KUKA KRL program: exC126.src, exC126.dat

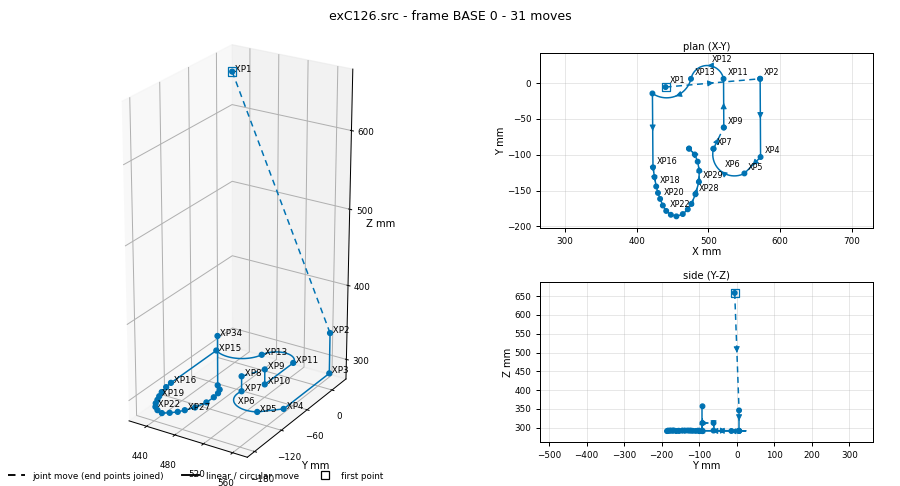
[picture p0: tool path of exC126.src in frame BASE 0, 31 of 33 moves have a stored position in this frame; points joined in program order, loops and branches not executed]
--- exC126.src ---
&ACCESS RVP
&REL 41
&PARAM EDITMASK = *
&PARAM TEMPLATE = C:\KRC\Roboter\Template\vorgabe
&PARAM DISKPATH = KRC:\R1\Program\126PARCIAL
DEF exC126( )
;FOLD INI;%{PE}
  ;FOLD BASISTECH INI
    GLOBAL INTERRUPT DECL 3 WHEN $STOPMESS==TRUE DO IR_STOPM ( )
    INTERRUPT ON 3
    BAS (#INITMOV,0 )
  ;ENDFOLD (BASISTECH INI)
  ;FOLD USER INI
    ;Make your modifications here

  ;ENDFOLD (USER INI)
;ENDFOLD (INI)

;FOLD SPTP HOME Vel=100 % DEFAULT ;%{PE}
;FOLD Parameters ;%{h}
;Params IlfProvider=kukaroboter.basistech.inlineforms.movement.spline; Kuka.IsGlobalPoint=False; Kuka.PointName=HOME; Kuka.BlendingEnabled=False; Kuka.MoveDataPtpName=DEFAULT; Kuka.VelocityPtp=100; Kuka.VelocityFieldEnabled=True; Kuka.CurrentCDSetIndex=0; Kuka.MovementParameterFieldEnabled=True; IlfCommand=SPTP
;ENDFOLD
SPTP XHOME WITH $VEL_AXIS[1] = SVEL_JOINT(100.0), $TOOL = STOOL2(FHOME), $BASE = SBASE(FHOME.BASE_NO), $IPO_MODE = SIPO_MODE(FHOME.IPO_FRAME), $LOAD = SLOAD(FHOME.TOOL_NO), $ACC_AXIS[1] = SACC_JOINT(PDEFAULT), $APO = SAPO_PTP(PDEFAULT), $GEAR_JERK[1] = SGEAR_JERK(PDEFAULT), $COLLMON_TOL_PRO[1] = USE_CM_PRO_VALUES(0)
;ENDFOLD

;FOLD SPTP P1 Vel=100 % PDAT1 Tool[1]:SMC Base[0] ;%{PE}
;FOLD Parameters ;%{h}
;Params IlfProvider=kukaroboter.basistech.inlineforms.movement.spline; Kuka.IsGlobalPoint=False; Kuka.PointName=P1; Kuka.BlendingEnabled=False; Kuka.MoveDataPtpName=PDAT1; Kuka.VelocityPtp=100; Kuka.VelocityFieldEnabled=True; Kuka.ColDetectFieldEnabled=True; Kuka.CurrentCDSetIndex=0; Kuka.MovementParameterFieldEnabled=True; IlfCommand=SPTP
;ENDFOLD
SPTP XP1 WITH $VEL_AXIS[1] = SVEL_JOINT(100.0), $TOOL = STOOL2(FP1), $BASE = SBASE(FP1.BASE_NO), $IPO_MODE = SIPO_MODE(FP1.IPO_FRAME), $LOAD = SLOAD(FP1.TOOL_NO), $ACC_AXIS[1] = SACC_JOINT(PPDAT1), $APO = SAPO_PTP(PPDAT1), $GEAR_JERK[1] = SGEAR_JERK(PPDAT1), $COLLMON_TOL_PRO[1] = USE_CM_PRO_VALUES(0)
;ENDFOLD
;FOLD SPTP P2 Vel=100 % PDAT2 Tool[1]:SMC Base[0] ;%{PE}
;FOLD Parameters ;%{h}
;Params IlfProvider=kukaroboter.basistech.inlineforms.movement.spline; Kuka.IsGlobalPoint=False; Kuka.PointName=P2; Kuka.BlendingEnabled=False; Kuka.MoveDataPtpName=PDAT2; Kuka.VelocityPtp=100; Kuka.VelocityFieldEnabled=True; Kuka.ColDetectFieldEnabled=True; Kuka.CurrentCDSetIndex=0; Kuka.MovementParameterFieldEnabled=True; IlfCommand=SPTP
;ENDFOLD
SPTP XP2 WITH $VEL_AXIS[1] = SVEL_JOINT(100.0), $TOOL = STOOL2(FP2), $BASE = SBASE(FP2.BASE_NO), $IPO_MODE = SIPO_MODE(FP2.IPO_FRAME), $LOAD = SLOAD(FP2.TOOL_NO), $ACC_AXIS[1] = SACC_JOINT(PPDAT2), $APO = SAPO_PTP(PPDAT2), $GEAR_JERK[1] = SGEAR_JERK(PPDAT2), $COLLMON_TOL_PRO[1] = USE_CM_PRO_VALUES(0)
;ENDFOLD
;FOLD SLIN P3 Vel=2 m/s CPDAT1 Tool[1]:SMC Base[0] ;%{PE}
;FOLD Parameters ;%{h}
;Params IlfProvider=kukaroboter.basistech.inlineforms.movement.spline; Kuka.IsGlobalPoint=False; Kuka.PointName=P3; Kuka.BlendingEnabled=False; Kuka.MoveDataName=CPDAT1; Kuka.VelocityPath=2; Kuka.VelocityFieldEnabled=True; Kuka.ColDetectFieldEnabled=True; Kuka.CurrentCDSetIndex=0; Kuka.MovementParameterFieldEnabled=True; IlfCommand=SLIN
;ENDFOLD
SLIN XP3 WITH $VEL = SVEL_CP(2.0, , LCPDAT1), $TOOL = STOOL2(FP3), $BASE = SBASE(FP3.BASE_NO), $IPO_MODE = SIPO_MODE(FP3.IPO_FRAME), $LOAD = SLOAD(FP3.TOOL_NO), $ACC = SACC_CP(LCPDAT1), $ORI_TYPE = SORI_TYP(LCPDAT1), $APO = SAPO(LCPDAT1), $JERK = SJERK(LCPDAT1), $COLLMON_TOL_PRO[1] = USE_CM_PRO_VALUES(0)
;ENDFOLD
;FOLD SLIN P4 Vel=2 m/s CPDAT2 Tool[1]:SMC Base[0] ;%{PE}
;FOLD Parameters ;%{h}
;Params IlfProvider=kukaroboter.basistech.inlineforms.movement.spline; Kuka.IsGlobalPoint=False; Kuka.PointName=P4; Kuka.BlendingEnabled=False; Kuka.MoveDataName=CPDAT2; Kuka.VelocityPath=2; Kuka.VelocityFieldEnabled=True; Kuka.ColDetectFieldEnabled=True; Kuka.CurrentCDSetIndex=0; Kuka.MovementParameterFieldEnabled=True; IlfCommand=SLIN
;ENDFOLD
SLIN XP4 WITH $VEL = SVEL_CP(2.0, , LCPDAT2), $TOOL = STOOL2(FP4), $BASE = SBASE(FP4.BASE_NO), $IPO_MODE = SIPO_MODE(FP4.IPO_FRAME), $LOAD = SLOAD(FP4.TOOL_NO), $ACC = SACC_CP(LCPDAT2), $ORI_TYPE = SORI_TYP(LCPDAT2), $APO = SAPO(LCPDAT2), $JERK = SJERK(LCPDAT2), $COLLMON_TOL_PRO[1] = USE_CM_PRO_VALUES(0)
;ENDFOLD
;FOLD SLIN P5 Vel=2 m/s CPDAT3 Tool[1]:SMC Base[0] ;%{PE}
;FOLD Parameters ;%{h}
;Params IlfProvider=kukaroboter.basistech.inlineforms.movement.spline; Kuka.IsGlobalPoint=False; Kuka.PointName=P5; Kuka.BlendingEnabled=False; Kuka.MoveDataName=CPDAT3; Kuka.VelocityPath=2; Kuka.VelocityFieldEnabled=True; Kuka.ColDetectFieldEnabled=True; Kuka.CurrentCDSetIndex=0; Kuka.MovementParameterFieldEnabled=True; IlfCommand=SLIN
;ENDFOLD
SLIN XP5 WITH $VEL = SVEL_CP(2.0, , LCPDAT3), $TOOL = STOOL2(FP5), $BASE = SBASE(FP5.BASE_NO), $IPO_MODE = SIPO_MODE(FP5.IPO_FRAME), $LOAD = SLOAD(FP5.TOOL_NO), $ACC = SACC_CP(LCPDAT3), $ORI_TYPE = SORI_TYP(LCPDAT3), $APO = SAPO(LCPDAT3), $JERK = SJERK(LCPDAT3), $COLLMON_TOL_PRO[1] = USE_CM_PRO_VALUES(0)
;ENDFOLD
;FOLD SCIRC P6 P7 Vel=2 m/s CPDAT4 Tool[1]:SMC Base[0] ;%{PE}
;FOLD Parameters ;%{h}
;Params IlfProvider=kukaroboter.basistech.inlineforms.movement.spline; Kuka.IsGlobalPoint=False; Kuka.PointName=P7; Kuka.HelpPointName=P6; Kuka.BlendingEnabled=False; Kuka.MoveDataName=CPDAT4; Kuka.VelocityPath=2; Kuka.VelocityFieldEnabled=True; Kuka.ColDetectFieldEnabled=True; Kuka.CurrentCDSetIndex=0; Kuka.MovementParameterFieldEnabled=True; IlfCommand=SCIRC
;ENDFOLD
SCIRC XP6, XP7 WITH $VEL = SVEL_CP(2.0, , LCPDAT4), $TOOL = STOOL2(FP7), $BASE = SBASE(FP7.BASE_NO), $IPO_MODE = SIPO_MODE(FP7.IPO_FRAME), $LOAD = SLOAD(FP7.TOOL_NO), $ACC = SACC_CP(LCPDAT4), $ORI_TYPE = SORI_TYP(LCPDAT4), $CIRC_TYPE = SCIRC_TYP(LCPDAT4), $APO = SAPO(LCPDAT4), $CIRC_MODE = SCIRC_M(LCPDAT4), $JERK = SJERK(LCPDAT4), $COLLMON_TOL_PRO[1] = USE_CM_PRO_VALUES(0)
;ENDFOLD
;FOLD SLIN P8 Vel=2 m/s CPDAT5 Tool[1]:SMC Base[0] ;%{PE}
;FOLD Parameters ;%{h}
;Params IlfProvider=kukaroboter.basistech.inlineforms.movement.spline; Kuka.IsGlobalPoint=False; Kuka.PointName=P8; Kuka.BlendingEnabled=False; Kuka.MoveDataName=CPDAT5; Kuka.VelocityPath=2; Kuka.VelocityFieldEnabled=True; Kuka.ColDetectFieldEnabled=True; Kuka.CurrentCDSetIndex=0; Kuka.MovementParameterFieldEnabled=True; IlfCommand=SLIN
;ENDFOLD
SLIN XP8 WITH $VEL = SVEL_CP(2.0, , LCPDAT5), $TOOL = STOOL2(FP8), $BASE = SBASE(FP8.BASE_NO), $IPO_MODE = SIPO_MODE(FP8.IPO_FRAME), $LOAD = SLOAD(FP8.TOOL_NO), $ACC = SACC_CP(LCPDAT5), $ORI_TYPE = SORI_TYP(LCPDAT5), $APO = SAPO(LCPDAT5), $JERK = SJERK(LCPDAT5), $COLLMON_TOL_PRO[1] = USE_CM_PRO_VALUES(0)
;ENDFOLD
;FOLD SPTP P9 Vel=100 % PDAT3 Tool[1]:SMC Base[0] ;%{PE}
;FOLD Parameters ;%{h}
;Params IlfProvider=kukaroboter.basistech.inlineforms.movement.spline; Kuka.IsGlobalPoint=False; Kuka.PointName=P9; Kuka.BlendingEnabled=False; Kuka.MoveDataPtpName=PDAT3; Kuka.VelocityPtp=100; Kuka.VelocityFieldEnabled=True; Kuka.ColDetectFieldEnabled=True; Kuka.CurrentCDSetIndex=0; Kuka.MovementParameterFieldEnabled=True; IlfCommand=SPTP
;ENDFOLD
SPTP XP9 WITH $VEL_AXIS[1] = SVEL_JOINT(100.0), $TOOL = STOOL2(FP9), $BASE = SBASE(FP9.BASE_NO), $IPO_MODE = SIPO_MODE(FP9.IPO_FRAME), $LOAD = SLOAD(FP9.TOOL_NO), $ACC_AXIS[1] = SACC_JOINT(PPDAT3), $APO = SAPO_PTP(PPDAT3), $GEAR_JERK[1] = SGEAR_JERK(PPDAT3), $COLLMON_TOL_PRO[1] = USE_CM_PRO_VALUES(0)
;ENDFOLD
;FOLD SLIN P10 Vel=2 m/s CPDAT6 Tool[1]:SMC Base[0] ;%{PE}
;FOLD Parameters ;%{h}
;Params IlfProvider=kukaroboter.basistech.inlineforms.movement.spline; Kuka.IsGlobalPoint=False; Kuka.PointName=P10; Kuka.BlendingEnabled=False; Kuka.MoveDataName=CPDAT6; Kuka.VelocityPath=2; Kuka.VelocityFieldEnabled=True; Kuka.ColDetectFieldEnabled=True; Kuka.CurrentCDSetIndex=0; Kuka.MovementParameterFieldEnabled=True; IlfCommand=SLIN
;ENDFOLD
SLIN XP10 WITH $VEL = SVEL_CP(2.0, , LCPDAT6), $TOOL = STOOL2(FP10), $BASE = SBASE(FP10.BASE_NO), $IPO_MODE = SIPO_MODE(FP10.IPO_FRAME), $LOAD = SLOAD(FP10.TOOL_NO), $ACC = SACC_CP(LCPDAT6), $ORI_TYPE = SORI_TYP(LCPDAT6), $APO = SAPO(LCPDAT6), $JERK = SJERK(LCPDAT6), $COLLMON_TOL_PRO[1] = USE_CM_PRO_VALUES(0)
;ENDFOLD
;FOLD SLIN P11 Vel=2 m/s CPDAT7 Tool[1]:SMC Base[0] ;%{PE}
;FOLD Parameters ;%{h}
;Params IlfProvider=kukaroboter.basistech.inlineforms.movement.spline; Kuka.IsGlobalPoint=False; Kuka.PointName=P11; Kuka.BlendingEnabled=False; Kuka.MoveDataName=CPDAT7; Kuka.VelocityPath=2; Kuka.VelocityFieldEnabled=True; Kuka.ColDetectFieldEnabled=True; Kuka.CurrentCDSetIndex=0; Kuka.MovementParameterFieldEnabled=True; IlfCommand=SLIN
;ENDFOLD
SLIN XP11 WITH $VEL = SVEL_CP(2.0, , LCPDAT7), $TOOL = STOOL2(FP11), $BASE = SBASE(FP11.BASE_NO), $IPO_MODE = SIPO_MODE(FP11.IPO_FRAME), $LOAD = SLOAD(FP11.TOOL_NO), $ACC = SACC_CP(LCPDAT7), $ORI_TYPE = SORI_TYP(LCPDAT7), $APO = SAPO(LCPDAT7), $JERK = SJERK(LCPDAT7), $COLLMON_TOL_PRO[1] = USE_CM_PRO_VALUES(0)
;ENDFOLD
;FOLD SCIRC P12 P13 Vel=2 m/s CPDAT8 Tool[1]:SMC Base[0] ;%{PE}
;FOLD Parameters ;%{h}
;Params IlfProvider=kukaroboter.basistech.inlineforms.movement.spline; Kuka.IsGlobalPoint=False; Kuka.PointName=P13; Kuka.HelpPointName=P12; Kuka.BlendingEnabled=False; Kuka.MoveDataName=CPDAT8; Kuka.VelocityPath=2; Kuka.VelocityFieldEnabled=True; Kuka.ColDetectFieldEnabled=True; Kuka.CurrentCDSetIndex=0; Kuka.MovementParameterFieldEnabled=True; IlfCommand=SCIRC
;ENDFOLD
SCIRC XP12, XP13 WITH $VEL = SVEL_CP(2.0, , LCPDAT8), $TOOL = STOOL2(FP13), $BASE = SBASE(FP13.BASE_NO), $IPO_MODE = SIPO_MODE(FP13.IPO_FRAME), $LOAD = SLOAD(FP13.TOOL_NO), $ACC = SACC_CP(LCPDAT8), $ORI_TYPE = SORI_TYP(LCPDAT8), $CIRC_TYPE = SCIRC_TYP(LCPDAT8), $APO = SAPO(LCPDAT8), $CIRC_MODE = SCIRC_M(LCPDAT8), $JERK = SJERK(LCPDAT8), $COLLMON_TOL_PRO[1] = USE_CM_PRO_VALUES(0)
;ENDFOLD
;FOLD SCIRC P14 P15 Vel=2 m/s CPDAT9 Tool[1]:SMC Base[0] ;%{PE}
;FOLD Parameters ;%{h}
;Params IlfProvider=kukaroboter.basistech.inlineforms.movement.spline; Kuka.IsGlobalPoint=False; Kuka.PointName=P15; Kuka.HelpPointName=P14; Kuka.BlendingEnabled=False; Kuka.MoveDataName=CPDAT9; Kuka.VelocityPath=2; Kuka.VelocityFieldEnabled=True; Kuka.ColDetectFieldEnabled=True; Kuka.CurrentCDSetIndex=0; Kuka.MovementParameterFieldEnabled=True; IlfCommand=SCIRC
;ENDFOLD
SCIRC XP14, XP15 WITH $VEL = SVEL_CP(2.0, , LCPDAT9), $TOOL = STOOL2(FP15), $BASE = SBASE(FP15.BASE_NO), $IPO_MODE = SIPO_MODE(FP15.IPO_FRAME), $LOAD = SLOAD(FP15.TOOL_NO), $ACC = SACC_CP(LCPDAT9), $ORI_TYPE = SORI_TYP(LCPDAT9), $CIRC_TYPE = SCIRC_TYP(LCPDAT9), $APO = SAPO(LCPDAT9), $CIRC_MODE = SCIRC_M(LCPDAT9), $JERK = SJERK(LCPDAT9), $COLLMON_TOL_PRO[1] = USE_CM_PRO_VALUES(0)
;ENDFOLD
;FOLD SLIN P16 Vel=2 m/s CPDAT10 Tool[1]:SMC Base[0] ;%{PE}
;FOLD Parameters ;%{h}
;Params IlfProvider=kukaroboter.basistech.inlineforms.movement.spline; Kuka.IsGlobalPoint=False; Kuka.PointName=P16; Kuka.BlendingEnabled=False; Kuka.MoveDataName=CPDAT10; Kuka.VelocityPath=2; Kuka.VelocityFieldEnabled=True; Kuka.ColDetectFieldEnabled=True; Kuka.CurrentCDSetIndex=0; Kuka.MovementParameterFieldEnabled=True; IlfCommand=SLIN
;ENDFOLD
SLIN XP16 WITH $VEL = SVEL_CP(2.0, , LCPDAT10), $TOOL = STOOL2(FP16), $BASE = SBASE(FP16.BASE_NO), $IPO_MODE = SIPO_MODE(FP16.IPO_FRAME), $LOAD = SLOAD(FP16.TOOL_NO), $ACC = SACC_CP(LCPDAT10), $ORI_TYPE = SORI_TYP(LCPDAT10), $APO = SAPO(LCPDAT10), $JERK = SJERK(LCPDAT10), $COLLMON_TOL_PRO[1] = USE_CM_PRO_VALUES(0)
;ENDFOLD
;FOLD SPLINE S1 Vel=2 m/s CPDAT11 Tool[1]:SMC Base[0] ;%{P} %CSPL_PARENT
;FOLD ;%{H}
;FOLD Parameters ;%{h}
;Params IlfProvider=kukaroboter.basistech.inlineforms.movement.splblock; Kuka.IsGlobalPoint=False; Kuka.SplineBlockPointName=S1; Kuka.BlendingEnabled=False; Kuka.MoveDataName=CPDAT11; Kuka.VelocityPath=2; Kuka.CurrentCDSetIndex=0; Kuka.MovementParameterFieldEnabled=True
;ENDFOLD
SPLINE WITH $VEL = SVEL_CP(2.0, , LCPDAT11), $TOOL = STOOL2(FS1), $BASE = SBASE(FS1.BASE_NO), $IPO_MODE = SIPO_MODE(FS1.IPO_FRAME), $LOAD = SLOAD(FS1.TOOL_NO), $ACC = SACC_CP(LCPDAT11), $APO = SAPO(LCPDAT11), $ORI_TYPE = SORI_TYP(LCPDAT11), $CIRC_TYPE = SCIRC_TYP(LCPDAT11), $JERK = SJERK(LCPDAT11), $COLLMON_TOL_PRO[1] = USE_CM_PRO_VALUES(0)
;ENDFOLD
;FOLD SPL P17 Vel=2 m/s CPDAT12 ColDetect= ;%{E}
;FOLD Parameters ;%{h}
;Params IlfProvider=kukaroboter.basistech.inlineforms.movement.spline; Kuka.IsGlobalPoint=False; Kuka.PointName=P17; Kuka.MoveDataName=CPDAT12; Kuka.VelocityPath=2; Kuka.VelocityFieldEnabled=True; Kuka.ColDetectFieldEnabled=True; Kuka.CurrentCDSetIndex=0; Kuka.MovementParameterFieldEnabled=True; IlfCommand=SPL
;ENDFOLD
SPL XP17 WITH $VEL = SVEL_CP(2.0, , LCPDAT12), $ACC = SACC_CP(LCPDAT12), $ORI_TYPE = SORI_TYP(LCPDAT12), $EX_AX_IGNORE = S_EXAX_IGN(LCPDAT12), $JERK = SJERK(LCPDAT12), $COLLMON_TOL_PRO[1] = USE_CM_PRO_VALUES(0)
;ENDFOLD
;FOLD SPL P18 Vel=2 m/s CPDAT13 ColDetect= ;%{E}
;FOLD Parameters ;%{h}
;Params IlfProvider=kukaroboter.basistech.inlineforms.movement.spline; Kuka.IsGlobalPoint=False; Kuka.PointName=P18; Kuka.MoveDataName=CPDAT13; Kuka.VelocityPath=2; Kuka.VelocityFieldEnabled=True; Kuka.ColDetectFieldEnabled=True; Kuka.CurrentCDSetIndex=0; Kuka.MovementParameterFieldEnabled=True; IlfCommand=SPL
;ENDFOLD
SPL XP18 WITH $VEL = SVEL_CP(2.0, , LCPDAT13), $ACC = SACC_CP(LCPDAT13), $ORI_TYPE = SORI_TYP(LCPDAT13), $EX_AX_IGNORE = S_EXAX_IGN(LCPDAT13), $JERK = SJERK(LCPDAT13), $COLLMON_TOL_PRO[1] = USE_CM_PRO_VALUES(0)
;ENDFOLD
;FOLD SPL P19 Vel=2 m/s CPDAT14 ColDetect= ;%{E}
;FOLD Parameters ;%{h}
;Params IlfProvider=kukaroboter.basistech.inlineforms.movement.spline; Kuka.IsGlobalPoint=False; Kuka.PointName=P19; Kuka.MoveDataName=CPDAT14; Kuka.VelocityPath=2; Kuka.VelocityFieldEnabled=True; Kuka.ColDetectFieldEnabled=True; Kuka.CurrentCDSetIndex=0; Kuka.MovementParameterFieldEnabled=True; IlfCommand=SPL
;ENDFOLD
SPL XP19 WITH $VEL = SVEL_CP(2.0, , LCPDAT14), $ACC = SACC_CP(LCPDAT14), $ORI_TYPE = SORI_TYP(LCPDAT14), $EX_AX_IGNORE = S_EXAX_IGN(LCPDAT14), $JERK = SJERK(LCPDAT14), $COLLMON_TOL_PRO[1] = USE_CM_PRO_VALUES(0)
;ENDFOLD
;FOLD SPL P20 Vel=2 m/s CPDAT15 ColDetect= ;%{E}
;FOLD Parameters ;%{h}
;Params IlfProvider=kukaroboter.basistech.inlineforms.movement.spline; Kuka.IsGlobalPoint=False; Kuka.PointName=P20; Kuka.MoveDataName=CPDAT15; Kuka.VelocityPath=2; Kuka.VelocityFieldEnabled=True; Kuka.ColDetectFieldEnabled=True; Kuka.CurrentCDSetIndex=0; Kuka.MovementParameterFieldEnabled=True; IlfCommand=SPL
;ENDFOLD
SPL XP20 WITH $VEL = SVEL_CP(2.0, , LCPDAT15), $ACC = SACC_CP(LCPDAT15), $ORI_TYPE = SORI_TYP(LCPDAT15), $EX_AX_IGNORE = S_EXAX_IGN(LCPDAT15), $JERK = SJERK(LCPDAT15), $COLLMON_TOL_PRO[1] = USE_CM_PRO_VALUES(0)
;ENDFOLD
;FOLD SPL P21 Vel=2 m/s CPDAT16 ColDetect= ;%{E}
;FOLD Parameters ;%{h}
;Params IlfProvider=kukaroboter.basistech.inlineforms.movement.spline; Kuka.IsGlobalPoint=False; Kuka.PointName=P21; Kuka.MoveDataName=CPDAT16; Kuka.VelocityPath=2; Kuka.VelocityFieldEnabled=True; Kuka.ColDetectFieldEnabled=True; Kuka.CurrentCDSetIndex=0; Kuka.MovementParameterFieldEnabled=True; IlfCommand=SPL
;ENDFOLD
SPL XP21 WITH $VEL = SVEL_CP(2.0, , LCPDAT16), $ACC = SACC_CP(LCPDAT16), $ORI_TYPE = SORI_TYP(LCPDAT16), $EX_AX_IGNORE = S_EXAX_IGN(LCPDAT16), $JERK = SJERK(LCPDAT16), $COLLMON_TOL_PRO[1] = USE_CM_PRO_VALUES(0)
;ENDFOLD
;FOLD SPL P22 Vel=2 m/s CPDAT17 ColDetect= ;%{E}
;FOLD Parameters ;%{h}
;Params IlfProvider=kukaroboter.basistech.inlineforms.movement.spline; Kuka.IsGlobalPoint=False; Kuka.PointName=P22; Kuka.MoveDataName=CPDAT17; Kuka.VelocityPath=2; Kuka.VelocityFieldEnabled=True; Kuka.ColDetectFieldEnabled=True; Kuka.CurrentCDSetIndex=0; Kuka.MovementParameterFieldEnabled=True; IlfCommand=SPL
;ENDFOLD
SPL XP22 WITH $VEL = SVEL_CP(2.0, , LCPDAT17), $ACC = SACC_CP(LCPDAT17), $ORI_TYPE = SORI_TYP(LCPDAT17), $EX_AX_IGNORE = S_EXAX_IGN(LCPDAT17), $JERK = SJERK(LCPDAT17), $COLLMON_TOL_PRO[1] = USE_CM_PRO_VALUES(0)
;ENDFOLD
;FOLD SPL P23 Vel=2 m/s CPDAT18 ColDetect= ;%{E}
;FOLD Parameters ;%{h}
;Params IlfProvider=kukaroboter.basistech.inlineforms.movement.spline; Kuka.IsGlobalPoint=False; Kuka.PointName=P23; Kuka.MoveDataName=CPDAT18; Kuka.VelocityPath=2; Kuka.VelocityFieldEnabled=True; Kuka.ColDetectFieldEnabled=True; Kuka.CurrentCDSetIndex=0; Kuka.MovementParameterFieldEnabled=True; IlfCommand=SPL
;ENDFOLD
SPL XP23 WITH $VEL = SVEL_CP(2.0, , LCPDAT18), $ACC = SACC_CP(LCPDAT18), $ORI_TYPE = SORI_TYP(LCPDAT18), $EX_AX_IGNORE = S_EXAX_IGN(LCPDAT18), $JERK = SJERK(LCPDAT18), $COLLMON_TOL_PRO[1] = USE_CM_PRO_VALUES(0)
;ENDFOLD
;FOLD SPL P24 Vel=2 m/s CPDAT19 ColDetect= ;%{E}
;FOLD Parameters ;%{h}
;Params IlfProvider=kukaroboter.basistech.inlineforms.movement.spline; Kuka.IsGlobalPoint=False; Kuka.PointName=P24; Kuka.MoveDataName=CPDAT19; Kuka.VelocityPath=2; Kuka.VelocityFieldEnabled=True; Kuka.ColDetectFieldEnabled=True; Kuka.CurrentCDSetIndex=0; Kuka.MovementParameterFieldEnabled=True; IlfCommand=SPL
;ENDFOLD
SPL XP24 WITH $VEL = SVEL_CP(2.0, , LCPDAT19), $ACC = SACC_CP(LCPDAT19), $ORI_TYPE = SORI_TYP(LCPDAT19), $EX_AX_IGNORE = S_EXAX_IGN(LCPDAT19), $JERK = SJERK(LCPDAT19), $COLLMON_TOL_PRO[1] = USE_CM_PRO_VALUES(0)
;ENDFOLD
;FOLD SPL P25 Vel=2 m/s CPDAT20 ColDetect= ;%{E}
;FOLD Parameters ;%{h}
;Params IlfProvider=kukaroboter.basistech.inlineforms.movement.spline; Kuka.IsGlobalPoint=False; Kuka.PointName=P25; Kuka.MoveDataName=CPDAT20; Kuka.VelocityPath=2; Kuka.VelocityFieldEnabled=True; Kuka.ColDetectFieldEnabled=True; Kuka.CurrentCDSetIndex=0; Kuka.MovementParameterFieldEnabled=True; IlfCommand=SPL
;ENDFOLD
SPL XP25 WITH $VEL = SVEL_CP(2.0, , LCPDAT20), $ACC = SACC_CP(LCPDAT20), $ORI_TYPE = SORI_TYP(LCPDAT20), $EX_AX_IGNORE = S_EXAX_IGN(LCPDAT20), $JERK = SJERK(LCPDAT20), $COLLMON_TOL_PRO[1] = USE_CM_PRO_VALUES(0)
;ENDFOLD
;FOLD SPL P26 Vel=2 m/s CPDAT21 ColDetect= ;%{E}
;FOLD Parameters ;%{h}
;Params IlfProvider=kukaroboter.basistech.inlineforms.movement.spline; Kuka.IsGlobalPoint=False; Kuka.PointName=P26; Kuka.MoveDataName=CPDAT21; Kuka.VelocityPath=2; Kuka.VelocityFieldEnabled=True; Kuka.ColDetectFieldEnabled=True; Kuka.CurrentCDSetIndex=0; Kuka.MovementParameterFieldEnabled=True; IlfCommand=SPL
;ENDFOLD
SPL XP26 WITH $VEL = SVEL_CP(2.0, , LCPDAT21), $ACC = SACC_CP(LCPDAT21), $ORI_TYPE = SORI_TYP(LCPDAT21), $EX_AX_IGNORE = S_EXAX_IGN(LCPDAT21), $JERK = SJERK(LCPDAT21), $COLLMON_TOL_PRO[1] = USE_CM_PRO_VALUES(0)
;ENDFOLD
;FOLD SPL P27 Vel=2 m/s CPDAT22 ColDetect= ;%{E}
;FOLD Parameters ;%{h}
;Params IlfProvider=kukaroboter.basistech.inlineforms.movement.spline; Kuka.IsGlobalPoint=False; Kuka.PointName=P27; Kuka.MoveDataName=CPDAT22; Kuka.VelocityPath=2; Kuka.VelocityFieldEnabled=True; Kuka.ColDetectFieldEnabled=True; Kuka.CurrentCDSetIndex=0; Kuka.MovementParameterFieldEnabled=True; IlfCommand=SPL
;ENDFOLD
SPL XP27 WITH $VEL = SVEL_CP(2.0, , LCPDAT22), $ACC = SACC_CP(LCPDAT22), $ORI_TYPE = SORI_TYP(LCPDAT22), $EX_AX_IGNORE = S_EXAX_IGN(LCPDAT22), $JERK = SJERK(LCPDAT22), $COLLMON_TOL_PRO[1] = USE_CM_PRO_VALUES(0)
;ENDFOLD
;FOLD SPL P28 Vel=2 m/s CPDAT23 ColDetect= ;%{E}
;FOLD Parameters ;%{h}
;Params IlfProvider=kukaroboter.basistech.inlineforms.movement.spline; Kuka.IsGlobalPoint=False; Kuka.PointName=P28; Kuka.MoveDataName=CPDAT23; Kuka.VelocityPath=2; Kuka.VelocityFieldEnabled=True; Kuka.ColDetectFieldEnabled=True; Kuka.CurrentCDSetIndex=0; Kuka.MovementParameterFieldEnabled=True; IlfCommand=SPL
;ENDFOLD
SPL XP28 WITH $VEL = SVEL_CP(2.0, , LCPDAT23), $ACC = SACC_CP(LCPDAT23), $ORI_TYPE = SORI_TYP(LCPDAT23), $EX_AX_IGNORE = S_EXAX_IGN(LCPDAT23), $JERK = SJERK(LCPDAT23), $COLLMON_TOL_PRO[1] = USE_CM_PRO_VALUES(0)
;ENDFOLD
;FOLD SPL P29 Vel=2 m/s CPDAT24 ColDetect= ;%{E}
;FOLD Parameters ;%{h}
;Params IlfProvider=kukaroboter.basistech.inlineforms.movement.spline; Kuka.IsGlobalPoint=False; Kuka.PointName=P29; Kuka.MoveDataName=CPDAT24; Kuka.VelocityPath=2; Kuka.VelocityFieldEnabled=True; Kuka.ColDetectFieldEnabled=True; Kuka.CurrentCDSetIndex=0; Kuka.MovementParameterFieldEnabled=True; IlfCommand=SPL
;ENDFOLD
SPL XP29 WITH $VEL = SVEL_CP(2.0, , LCPDAT24), $ACC = SACC_CP(LCPDAT24), $ORI_TYPE = SORI_TYP(LCPDAT24), $EX_AX_IGNORE = S_EXAX_IGN(LCPDAT24), $JERK = SJERK(LCPDAT24), $COLLMON_TOL_PRO[1] = USE_CM_PRO_VALUES(0)
;ENDFOLD
;FOLD SPL P30 Vel=2 m/s CPDAT25 ColDetect= ;%{E}
;FOLD Parameters ;%{h}
;Params IlfProvider=kukaroboter.basistech.inlineforms.movement.spline; Kuka.IsGlobalPoint=False; Kuka.PointName=P30; Kuka.MoveDataName=CPDAT25; Kuka.VelocityPath=2; Kuka.VelocityFieldEnabled=True; Kuka.ColDetectFieldEnabled=True; Kuka.CurrentCDSetIndex=0; Kuka.MovementParameterFieldEnabled=True; IlfCommand=SPL
;ENDFOLD
SPL XP30 WITH $VEL = SVEL_CP(2.0, , LCPDAT25), $ACC = SACC_CP(LCPDAT25), $ORI_TYPE = SORI_TYP(LCPDAT25), $EX_AX_IGNORE = S_EXAX_IGN(LCPDAT25), $JERK = SJERK(LCPDAT25), $COLLMON_TOL_PRO[1] = USE_CM_PRO_VALUES(0)
;ENDFOLD
;FOLD SPL P31 Vel=2 m/s CPDAT26 ColDetect= ;%{E}
;FOLD Parameters ;%{h}
;Params IlfProvider=kukaroboter.basistech.inlineforms.movement.spline; Kuka.IsGlobalPoint=False; Kuka.PointName=P31; Kuka.MoveDataName=CPDAT26; Kuka.VelocityPath=2; Kuka.VelocityFieldEnabled=True; Kuka.ColDetectFieldEnabled=True; Kuka.CurrentCDSetIndex=0; Kuka.MovementParameterFieldEnabled=True; IlfCommand=SPL
;ENDFOLD
SPL XP31 WITH $VEL = SVEL_CP(2.0, , LCPDAT26), $ACC = SACC_CP(LCPDAT26), $ORI_TYPE = SORI_TYP(LCPDAT26), $EX_AX_IGNORE = S_EXAX_IGN(LCPDAT26), $JERK = SJERK(LCPDAT26), $COLLMON_TOL_PRO[1] = USE_CM_PRO_VALUES(0)
;ENDFOLD
;FOLD SPL P32 Vel=2 m/s CPDAT27 ColDetect= ;%{E}
;FOLD Parameters ;%{h}
;Params IlfProvider=kukaroboter.basistech.inlineforms.movement.spline; Kuka.IsGlobalPoint=False; Kuka.PointName=P32; Kuka.MoveDataName=CPDAT27; Kuka.VelocityPath=2; Kuka.VelocityFieldEnabled=True; Kuka.ColDetectFieldEnabled=True; Kuka.CurrentCDSetIndex=0; Kuka.MovementParameterFieldEnabled=True; IlfCommand=SPL
;ENDFOLD
SPL XP32 WITH $VEL = SVEL_CP(2.0, , LCPDAT27), $ACC = SACC_CP(LCPDAT27), $ORI_TYPE = SORI_TYP(LCPDAT27), $EX_AX_IGNORE = S_EXAX_IGN(LCPDAT27), $JERK = SJERK(LCPDAT27), $COLLMON_TOL_PRO[1] = USE_CM_PRO_VALUES(0)
;ENDFOLD
;FOLD SPL P33 Vel=2 m/s CPDAT28 ColDetect= ;%{E}
;FOLD Parameters ;%{h}
;Params IlfProvider=kukaroboter.basistech.inlineforms.movement.spline; Kuka.IsGlobalPoint=False; Kuka.PointName=P33; Kuka.MoveDataName=CPDAT28; Kuka.VelocityPath=2; Kuka.VelocityFieldEnabled=True; Kuka.ColDetectFieldEnabled=True; Kuka.CurrentCDSetIndex=0; Kuka.MovementParameterFieldEnabled=True; IlfCommand=SPL
;ENDFOLD
SPL XP33 WITH $VEL = SVEL_CP(2.0, , LCPDAT28), $ACC = SACC_CP(LCPDAT28), $ORI_TYPE = SORI_TYP(LCPDAT28), $EX_AX_IGNORE = S_EXAX_IGN(LCPDAT28), $JERK = SJERK(LCPDAT28), $COLLMON_TOL_PRO[1] = USE_CM_PRO_VALUES(0)
;ENDFOLD
;FOLD ;%{H}
ENDSPLINE
;ENDFOLD
;ENDFOLD ENDSPLINE ;%{V}

;FOLD SLIN P34 Vel=2 m/s CPDAT29 Tool[1]:SMC Base[0] ;%{PE}
;FOLD Parameters ;%{h}
;Params IlfProvider=kukaroboter.basistech.inlineforms.movement.spline; Kuka.IsGlobalPoint=False; Kuka.PointName=P34; Kuka.BlendingEnabled=False; Kuka.MoveDataName=CPDAT29; Kuka.VelocityPath=2; Kuka.VelocityFieldEnabled=True; Kuka.ColDetectFieldEnabled=True; Kuka.CurrentCDSetIndex=0; Kuka.MovementParameterFieldEnabled=True; IlfCommand=SLIN
;ENDFOLD
SLIN XP34 WITH $VEL = SVEL_CP(2.0, , LCPDAT29), $TOOL = STOOL2(FP34), $BASE = SBASE(FP34.BASE_NO), $IPO_MODE = SIPO_MODE(FP34.IPO_FRAME), $LOAD = SLOAD(FP34.TOOL_NO), $ACC = SACC_CP(LCPDAT29), $ORI_TYPE = SORI_TYP(LCPDAT29), $APO = SAPO(LCPDAT29), $JERK = SJERK(LCPDAT29), $COLLMON_TOL_PRO[1] = USE_CM_PRO_VALUES(0)
;ENDFOLD
;FOLD SPTP HOME Vel=100 % DEFAULT ;%{PE}
;FOLD Parameters ;%{h}
;Params IlfProvider=kukaroboter.basistech.inlineforms.movement.spline; Kuka.IsGlobalPoint=False; Kuka.PointName=HOME; Kuka.BlendingEnabled=False; Kuka.MoveDataPtpName=DEFAULT; Kuka.VelocityPtp=100; Kuka.VelocityFieldEnabled=True; Kuka.CurrentCDSetIndex=0; Kuka.MovementParameterFieldEnabled=True; IlfCommand=SPTP
;ENDFOLD
SPTP XHOME WITH $VEL_AXIS[1] = SVEL_JOINT(100.0), $TOOL = STOOL2(FHOME), $BASE = SBASE(FHOME.BASE_NO), $IPO_MODE = SIPO_MODE(FHOME.IPO_FRAME), $LOAD = SLOAD(FHOME.TOOL_NO), $ACC_AXIS[1] = SACC_JOINT(PDEFAULT), $APO = SAPO_PTP(PDEFAULT), $GEAR_JERK[1] = SGEAR_JERK(PDEFAULT), $COLLMON_TOL_PRO[1] = USE_CM_PRO_VALUES(0)
;ENDFOLD

END

--- exC126.dat ---
&ACCESS RVP
&REL 41
&PARAM EDITMASK = *
&PARAM TEMPLATE = C:\KRC\Roboter\Template\vorgabe
&PARAM DISKPATH = KRC:\R1\Program\126PARCIAL
DEFDAT  exC126
;FOLD EXTERNAL DECLARATIONS;%{PE}%MKUKATPBASIS,%CEXT,%VCOMMON,%P
;FOLD BASISTECH EXT;%{PE}%MKUKATPBASIS,%CEXT,%VEXT,%P
EXT  BAS (BAS_COMMAND  :IN,REAL  :IN )
DECL INT SUCCESS
;ENDFOLD (BASISTECH EXT)
;FOLD USER EXT;%{E}%MKUKATPUSER,%CEXT,%VEXT,%P
;Make your modifications here

;ENDFOLD (USER EXT)
;ENDFOLD (EXTERNAL DECLARATIONS)
DECL E6POS XP1={X 440.254517,Y -5.46516228,Z 658.758850,A -91.4489288,B 89.2024460,C -90.6416245,S 2,T 34,E1 0.0,E2 0.0,E3 0.0,E4 0.0,E5 0.0,E6 0.0}
DECL FDAT FP1={TOOL_NO 1,BASE_NO 0,IPO_FRAME #BASE,POINT2[] " "}
DECL PDAT PPDAT1={VEL 100.000,ACC 100.000,APO_DIST 500.000,APO_MODE #CDIS,GEAR_JERK 100.000,EXAX_IGN 0}
DECL MODULEPARAM_T LAST_TP_PARAMS={PARAMS[] "Kuka.VelocityFieldEnabled=True; Kuka.ColDetectFieldEnabled=True; Kuka.MovementParameterFieldEnabled=True; Kuka.IsAngleEnabled=False; Kuka.PointName=P34; Kuka.FrameData.base_no=0; Kuka.FrameData.tool_no=1; Kuka.FrameData.ipo_frame=#BASE; Kuka.isglobalpoint=False; Kuka.MoveDataPtpName=PDAT3; Kuka.MovementDataPdat.apo_mode=#CDIS; Kuka.MovementDataPdat.apo_dist=500; Kuka.MovementData.vel=2; Kuka.MovementData.acc=100; Kuka.MovementData.gear_jerk=100; Kuka.MovementData.exax_ign=0; Kuka.VelocityPtp=100; Kuka.BlendingEnabled=False; Kuka.CurrentCDSetIndex=0; Kuka.MoveDataName=CPDAT29; Kuka.MovementData.apo_fac=50; Kuka.MovementData.apo_dist=500; Kuka.MovementData.axis_acc=100; Kuka.MovementData.axis_vel=100; Kuka.MovementData.circ_typ=#BASE; Kuka.MovementData.jerk_fac=50; Kuka.MovementData.ori_typ=#VAR; Kuka.VelocityPath=2; Kuka.MovementData.cb={AUX_PT {ORI #CONSIDER,E1 #CONSIDER,E2 #CONSIDER,E3 #CONSIDER,E4 #CONSIDER,E5 #CONSIDER,E6 #CONSIDER},TARGET_PT {ORI #INTERPOLATE,E1 #INTERPOLATE,E2 #INTERPOLATE,E3 #INTERPOLATE,E4 #INTERPOLATE,E5 #INTERPOLATE,E6 #INTERPOLATE}}; Kuka.HelpPointName=P14; Kuka.SplineBlockPointName=S1                                    "}
DECL E6POS XP2={X 572.217285,Y 6.13008738,Z 345.845581,A -91.2445374,B 89.2024460,C -90.6405869,S 2,T 35,E1 0.0,E2 0.0,E3 0.0,E4 0.0,E5 0.0,E6 0.0}
DECL FDAT FP2={TOOL_NO 1,BASE_NO 0,IPO_FRAME #BASE,POINT2[] " "}
DECL PDAT PPDAT2={VEL 100.000,ACC 100.000,APO_DIST 500.000,APO_MODE #CDIS,GEAR_JERK 100.000,EXAX_IGN 0}
DECL E6POS XP3={X 572.217285,Y 6.13008690,Z 291.103058,A -91.2445374,B 89.2024460,C -90.6405869,S 2,T 35,E1 0.0,E2 0.0,E3 0.0,E4 0.0,E5 0.0,E6 0.0}
DECL FDAT FP3={TOOL_NO 1,BASE_NO 0,IPO_FRAME #BASE,POINT2[] " "}
DECL LDAT LCPDAT1={VEL 2.00000,ACC 100.000,APO_DIST 500.000,APO_FAC 50.0000,AXIS_VEL 100.000,AXIS_ACC 100.000,ORI_TYP #VAR,CIRC_TYP #BASE,JERK_FAC 50.0000,GEAR_JERK 100.000,EXAX_IGN 0}
DECL E6POS XP4={X 572.820129,Y -103.115692,Z 291.908752,A -91.2445297,B 89.2024460,C -90.6405792,S 2,T 2,E1 0.0,E2 0.0,E3 0.0,E4 0.0,E5 0.0,E6 0.0}
DECL FDAT FP4={TOOL_NO 1,BASE_NO 0,IPO_FRAME #BASE,POINT2[] " "}
DECL LDAT LCPDAT2={VEL 2.00000,ACC 100.000,APO_DIST 500.000,APO_FAC 50.0000,AXIS_VEL 100.000,AXIS_ACC 100.000,ORI_TYP #VAR,CIRC_TYP #BASE,JERK_FAC 50.0000,GEAR_JERK 100.000,EXAX_IGN 0}
DECL E6POS XP5={X 550.268677,Y -125.986488,Z 291.847626,A -91.2445068,B 89.2024460,C -90.6405563,S 2,T 2,E1 0.0,E2 0.0,E3 0.0,E4 0.0,E5 0.0,E6 0.0}
DECL FDAT FP5={TOOL_NO 1,BASE_NO 0,IPO_FRAME #BASE,POINT2[] " "}
DECL LDAT LCPDAT3={VEL 2.00000,ACC 100.000,APO_DIST 500.000,APO_FAC 50.0000,AXIS_VEL 100.000,AXIS_ACC 100.000,ORI_TYP #VAR,CIRC_TYP #BASE,JERK_FAC 50.0000,GEAR_JERK 100.000,EXAX_IGN 0}
DECL E6POS XP6={X 516.915161,Y -122.442421,Z 291.819275,A -91.2192841,B 89.2022,C -90.6168823,S 2,T 2,E1 0.0,E2 0.0,E3 0.0,E4 0.0,E5 0.0,E6 0.0}
DECL E6POS XP7={X 507.097961,Y -91.5420761,Z 291.894928,A -91.2380219,B 89.2022552,C -90.6352768,S 2,T 2,E1 0.0,E2 0.0,E3 0.0,E4 0.0,E5 0.0,E6 0.0}
DECL FDAT FP7={TOOL_NO 1,BASE_NO 0,IPO_FRAME #BASE,POINT2[] " "}
DECL LDAT LCPDAT4={VEL 2.00000,ACC 100.000,APO_DIST 500.000,APO_FAC 50.0000,AXIS_VEL 100.000,AXIS_ACC 100.000,ORI_TYP #VAR,CIRC_TYP #BASE,JERK_FAC 50.0000,GEAR_JERK 100.000,EXAX_IGN 0,CB {AUX_PT {ORI #CONSIDER,E1 #CONSIDER,E2 #CONSIDER,E3 #CONSIDER,E4 #CONSIDER,E5 #CONSIDER,E6 #CONSIDER},TARGET_PT {ORI #INTERPOLATE,E1 #INTERPOLATE,E2 #INTERPOLATE,E3 #INTERPOLATE,E4 #INTERPOLATE,E5 #INTERPOLATE,E6 #INTERPOLATE}}}
DECL E6POS XP8={X 507.097961,Y -91.5420761,Z 312.081970,A -91.2380219,B 89.2022552,C -90.6352768,S 2,T 2,E1 0.0,E2 0.0,E3 0.0,E4 0.0,E5 0.0,E6 0.0}
DECL FDAT FP8={TOOL_NO 1,BASE_NO 0,IPO_FRAME #BASE,POINT2[] " "}
DECL LDAT LCPDAT5={VEL 2.00000,ACC 100.000,APO_DIST 500.000,APO_FAC 50.0000,AXIS_VEL 100.000,AXIS_ACC 100.000,ORI_TYP #VAR,CIRC_TYP #BASE,JERK_FAC 50.0000,GEAR_JERK 100.000,EXAX_IGN 0}
DECL E6POS XP9={X 521.494202,Y -61.8792267,Z 312.287628,A -91.2365341,B 89.2022552,C -90.6352463,S 2,T 2,E1 0.0,E2 0.0,E3 0.0,E4 0.0,E5 0.0,E6 0.0}
DECL FDAT FP9={TOOL_NO 1,BASE_NO 0,IPO_FRAME #BASE,POINT2[] " "}
DECL PDAT PPDAT3={VEL 100.000,ACC 100.000,APO_DIST 500.000,APO_MODE #CDIS,GEAR_JERK 100.000,EXAX_IGN 0}
DECL E6POS XP10={X 521.494202,Y -61.8792267,Z 292.015533,A -91.2365189,B 89.2022552,C -90.6352310,S 2,T 2,E1 0.0,E2 0.0,E3 0.0,E4 0.0,E5 0.0,E6 0.0}
DECL FDAT FP10={TOOL_NO 1,BASE_NO 0,IPO_FRAME #BASE,POINT2[] " "}
DECL LDAT LCPDAT6={VEL 2.00000,ACC 100.000,APO_DIST 500.000,APO_FAC 50.0000,AXIS_VEL 100.000,AXIS_ACC 100.000,ORI_TYP #VAR,CIRC_TYP #BASE,JERK_FAC 50.0000,GEAR_JERK 100.000,EXAX_IGN 0}
DECL E6POS XP11={X 521.153564,Y 6.04988909,Z 291.641907,A -91.2365,B 89.2022552,C -90.6352234,S 2,T 35,E1 0.0,E2 0.0,E3 0.0,E4 0.0,E5 0.0,E6 0.0}
DECL FDAT FP11={TOOL_NO 1,BASE_NO 0,IPO_FRAME #BASE,POINT2[] " "}
DECL LDAT LCPDAT7={VEL 2.00000,ACC 100.000,APO_DIST 500.000,APO_FAC 50.0000,AXIS_VEL 100.000,AXIS_ACC 100.000,ORI_TYP #VAR,CIRC_TYP #BASE,JERK_FAC 50.0000,GEAR_JERK 100.000,EXAX_IGN 0}
DECL E6POS XP12={X 499.559601,Y 24.6250229,Z 291.305359,A -91.2364883,B 89.2022552,C -90.6352,S 2,T 35,E1 0.0,E2 0.0,E3 0.0,E4 0.0,E5 0.0,E6 0.0}
DECL E6POS XP13={X 475.699707,Y 6.04398346,Z 290.662018,A -91.2364807,B 89.2022552,C -90.6351929,S 2,T 35,E1 0.0,E2 0.0,E3 0.0,E4 0.0,E5 0.0,E6 0.0}
DECL FDAT FP13={TOOL_NO 1,BASE_NO 0,IPO_FRAME #BASE,POINT2[] " "}
DECL LDAT LCPDAT8={VEL 2.00000,ACC 100.000,APO_DIST 500.000,APO_FAC 50.0000,AXIS_VEL 100.000,AXIS_ACC 100.000,ORI_TYP #VAR,CIRC_TYP #BASE,JERK_FAC 50.0000,GEAR_JERK 100.000,EXAX_IGN 0,CB {AUX_PT {ORI #CONSIDER,E1 #CONSIDER,E2 #CONSIDER,E3 #CONSIDER,E4 #CONSIDER,E5 #CONSIDER,E6 #CONSIDER},TARGET_PT {ORI #INTERPOLATE,E1 #INTERPOLATE,E2 #INTERPOLATE,E3 #INTERPOLATE,E4 #INTERPOLATE,E5 #INTERPOLATE,E6 #INTERPOLATE}}}
DECL E6POS XP14={X 453.690521,Y -18.3389587,Z 290.361481,A -91.2364655,B 89.2022552,C -90.6351776,S 2,T 34,E1 0.0,E2 0.0,E3 0.0,E4 0.0,E5 0.0,E6 0.0}
DECL E6POS XP15={X 421.889099,Y -14.3608494,Z 290.936707,A -91.2364426,B 89.2022552,C -90.6351547,S 2,T 34,E1 0.0,E2 0.0,E3 0.0,E4 0.0,E5 0.0,E6 0.0}
DECL FDAT FP15={TOOL_NO 1,BASE_NO 0,IPO_FRAME #BASE,POINT2[] " "}
DECL LDAT LCPDAT9={VEL 2.00000,ACC 100.000,APO_DIST 500.000,APO_FAC 50.0000,AXIS_VEL 100.000,AXIS_ACC 100.000,ORI_TYP #VAR,CIRC_TYP #BASE,JERK_FAC 50.0000,GEAR_JERK 100.000,EXAX_IGN 0,CB {AUX_PT {ORI #CONSIDER,E1 #CONSIDER,E2 #CONSIDER,E3 #CONSIDER,E4 #CONSIDER,E5 #CONSIDER,E6 #CONSIDER},TARGET_PT {ORI #INTERPOLATE,E1 #INTERPOLATE,E2 #INTERPOLATE,E3 #INTERPOLATE,E4 #INTERPOLATE,E5 #INTERPOLATE,E6 #INTERPOLATE}}}
DECL E6POS XP16={X 422.646729,Y -117.423416,Z 291.368103,A -90.7243652,B 89.2004929,C -90.1250916,S 2,T 2,E1 0.0,E2 0.0,E3 0.0,E4 0.0,E5 0.0,E6 0.0}
DECL FDAT FP16={TOOL_NO 1,BASE_NO 0,IPO_FRAME #BASE,POINT2[] " "}
DECL LDAT LCPDAT10={VEL 2.00000,ACC 100.000,APO_DIST 500.000,APO_FAC 50.0000,AXIS_VEL 100.000,AXIS_ACC 100.000,ORI_TYP #VAR,CIRC_TYP #BASE,JERK_FAC 50.0000,GEAR_JERK 100.000,EXAX_IGN 0}
DECL FDAT FS1={TOOL_NO 1,BASE_NO 0,IPO_FRAME #BASE,POINT2[] " "}
DECL LDAT LCPDAT11={VEL 2.00000,ACC 100.000,APO_DIST 500.000,APO_FAC 50.0000,AXIS_VEL 100.000,AXIS_ACC 100.000,ORI_TYP #VAR,CIRC_TYP #BASE,JERK_FAC 50.0000,GEAR_JERK 100.000,EXAX_IGN 0}
DECL E6POS XP17={X 424.784698,Y -131.035080,Z 292.182739,A -90.7243500,B 89.2004929,C -90.1250839,S 2,T 2,E1 0.0,E2 0.0,E3 0.0,E4 0.0,E5 0.0,E6 0.0}
DECL LDAT LCPDAT12={VEL 2.00000,ACC 100.000,APO_DIST 500.000,APO_FAC 50.0000,AXIS_VEL 100.000,AXIS_ACC 100.000,ORI_TYP #VAR,CIRC_TYP #BASE,JERK_FAC 50.0000,GEAR_JERK 100.000,EXAX_IGN 0}
DECL E6POS XP18={X 427.170166,Y -144.176315,Z 292.023224,A -90.7215500,B 89.2004929,C -90.1250687,S 2,T 2,E1 0.0,E2 0.0,E3 0.0,E4 0.0,E5 0.0,E6 0.0}
DECL LDAT LCPDAT13={VEL 2.00000,ACC 100.000,APO_DIST 500.000,APO_FAC 50.0000,AXIS_VEL 100.000,AXIS_ACC 100.000,ORI_TYP #VAR,CIRC_TYP #BASE,JERK_FAC 50.0000,GEAR_JERK 100.000,EXAX_IGN 0}
DECL E6POS XP19={X 429.624359,Y -153.201324,Z 291.151764,A -90.7215424,B 89.2004929,C -90.1250610,S 2,T 2,E1 0.0,E2 0.0,E3 0.0,E4 0.0,E5 0.0,E6 0.0}
DECL LDAT LCPDAT14={VEL 2.00000,ACC 100.000,APO_DIST 500.000,APO_FAC 50.0000,AXIS_VEL 100.000,AXIS_ACC 100.000,ORI_TYP #VAR,CIRC_TYP #BASE,JERK_FAC 50.0000,GEAR_JERK 100.000,EXAX_IGN 0}
DECL E6POS XP20={X 432.632202,Y -161.518051,Z 290.851166,A -90.7232056,B 89.2004929,C -90.1250534,S 2,T 2,E1 0.0,E2 0.0,E3 0.0,E4 0.0,E5 0.0,E6 0.0}
DECL LDAT LCPDAT15={VEL 2.00000,ACC 100.000,APO_DIST 500.000,APO_FAC 50.0000,AXIS_VEL 100.000,AXIS_ACC 100.000,ORI_TYP #VAR,CIRC_TYP #BASE,JERK_FAC 50.0000,GEAR_JERK 100.000,EXAX_IGN 0}
DECL E6POS XP21={X 436.401398,Y -170.746506,Z 291.407623,A -90.7231903,B 89.2004929,C -90.1250381,S 2,T 2,E1 0.0,E2 0.0,E3 0.0,E4 0.0,E5 0.0,E6 0.0}
DECL LDAT LCPDAT16={VEL 2.00000,ACC 100.000,APO_DIST 500.000,APO_FAC 50.0000,AXIS_VEL 100.000,AXIS_ACC 100.000,ORI_TYP #VAR,CIRC_TYP #BASE,JERK_FAC 50.0000,GEAR_JERK 100.000,EXAX_IGN 0}
DECL E6POS XP22={X 441.123535,Y -178.336746,Z 291.486694,A -90.7231750,B 89.2004929,C -90.1250229,S 2,T 2,E1 0.0,E2 0.0,E3 0.0,E4 0.0,E5 0.0,E6 0.0}
DECL LDAT LCPDAT17={VEL 2.00000,ACC 100.000,APO_DIST 500.000,APO_FAC 50.0000,AXIS_VEL 100.000,AXIS_ACC 100.000,ORI_TYP #VAR,CIRC_TYP #BASE,JERK_FAC 50.0000,GEAR_JERK 100.000,EXAX_IGN 0}
DECL E6POS XP23={X 447.589478,Y -183.696960,Z 291.271729,A -90.7231598,B 89.2004929,C -90.1250,S 2,T 2,E1 0.0,E2 0.0,E3 0.0,E4 0.0,E5 0.0,E6 0.0}
DECL LDAT LCPDAT18={VEL 2.00000,ACC 100.000,APO_DIST 500.000,APO_FAC 50.0000,AXIS_VEL 100.000,AXIS_ACC 100.000,ORI_TYP #VAR,CIRC_TYP #BASE,JERK_FAC 50.0000,GEAR_JERK 100.000,EXAX_IGN 0}
DECL E6POS XP24={X 455.333282,Y -185.901962,Z 290.563873,A -90.7231369,B 89.2004929,C -90.1249847,S 2,T 2,E1 0.0,E2 0.0,E3 0.0,E4 0.0,E5 0.0,E6 0.0}
DECL LDAT LCPDAT19={VEL 2.00000,ACC 100.000,APO_DIST 500.000,APO_FAC 50.0000,AXIS_VEL 100.000,AXIS_ACC 100.000,ORI_TYP #VAR,CIRC_TYP #BASE,JERK_FAC 50.0000,GEAR_JERK 100.000,EXAX_IGN 0}
DECL E6POS XP25={X 464.274597,Y -182.709122,Z 292.005829,A -90.7231216,B 89.2004929,C -90.1249695,S 2,T 2,E1 0.0,E2 0.0,E3 0.0,E4 0.0,E5 0.0,E6 0.0}
DECL LDAT LCPDAT20={VEL 2.00000,ACC 100.000,APO_DIST 500.000,APO_FAC 50.0000,AXIS_VEL 100.000,AXIS_ACC 100.000,ORI_TYP #VAR,CIRC_TYP #BASE,JERK_FAC 50.0000,GEAR_JERK 100.000,EXAX_IGN 0}
DECL E6POS XP26={X 471.236115,Y -176.090515,Z 292.286469,A -90.7231064,B 89.2004929,C -90.1249466,S 2,T 2,E1 0.0,E2 0.0,E3 0.0,E4 0.0,E5 0.0,E6 0.0}
DECL LDAT LCPDAT21={VEL 2.00000,ACC 100.000,APO_DIST 500.000,APO_FAC 50.0000,AXIS_VEL 100.000,AXIS_ACC 100.000,ORI_TYP #VAR,CIRC_TYP #BASE,JERK_FAC 50.0000,GEAR_JERK 100.000,EXAX_IGN 0}
DECL E6POS XP27={X 476.257751,Y -168.615845,Z 292.515228,A -90.7230911,B 89.2004929,C -90.1249390,S 2,T 2,E1 0.0,E2 0.0,E3 0.0,E4 0.0,E5 0.0,E6 0.0}
DECL LDAT LCPDAT22={VEL 2.00000,ACC 100.000,APO_DIST 500.000,APO_FAC 50.0000,AXIS_VEL 100.000,AXIS_ACC 100.000,ORI_TYP #VAR,CIRC_TYP #BASE,JERK_FAC 50.0000,GEAR_JERK 100.000,EXAX_IGN 0}
DECL E6POS XP28={X 481.917664,Y -155.092072,Z 291.616302,A -90.7230759,B 89.2004929,C -90.1249237,S 2,T 2,E1 0.0,E2 0.0,E3 0.0,E4 0.0,E5 0.0,E6 0.0}
DECL LDAT LCPDAT23={VEL 2.00000,ACC 100.000,APO_DIST 500.000,APO_FAC 50.0000,AXIS_VEL 100.000,AXIS_ACC 100.000,ORI_TYP #VAR,CIRC_TYP #BASE,JERK_FAC 50.0000,GEAR_JERK 100.000,EXAX_IGN 0}
DECL E6POS XP29={X 486.720062,Y -137.813339,Z 291.947357,A -90.7246704,B 89.1985931,C -90.1231842,S 2,T 2,E1 0.0,E2 0.0,E3 0.0,E4 0.0,E5 0.0,E6 0.0}
DECL LDAT LCPDAT24={VEL 2.00000,ACC 100.000,APO_DIST 500.000,APO_FAC 50.0000,AXIS_VEL 100.000,AXIS_ACC 100.000,ORI_TYP #VAR,CIRC_TYP #BASE,JERK_FAC 50.0000,GEAR_JERK 100.000,EXAX_IGN 0}
DECL E6POS XP30={X 487.248840,Y -122.315338,Z 292.028503,A -90.7246552,B 89.1985931,C -90.1231689,S 2,T 2,E1 0.0,E2 0.0,E3 0.0,E4 0.0,E5 0.0,E6 0.0}
DECL LDAT LCPDAT25={VEL 2.00000,ACC 100.000,APO_DIST 500.000,APO_FAC 50.0000,AXIS_VEL 100.000,AXIS_ACC 100.000,ORI_TYP #VAR,CIRC_TYP #BASE,JERK_FAC 50.0000,GEAR_JERK 100.000,EXAX_IGN 0}
DECL E6POS XP31={X 485.048523,Y -109.539658,Z 291.113922,A -90.7246475,B 89.1985931,C -90.1231613,S 2,T 2,E1 0.0,E2 0.0,E3 0.0,E4 0.0,E5 0.0,E6 0.0}
DECL LDAT LCPDAT26={VEL 2.00000,ACC 100.000,APO_DIST 500.000,APO_FAC 50.0000,AXIS_VEL 100.000,AXIS_ACC 100.000,ORI_TYP #VAR,CIRC_TYP #BASE,JERK_FAC 50.0000,GEAR_JERK 100.000,EXAX_IGN 0}
DECL E6POS XP32={X 480.979797,Y -99.5248108,Z 290.458191,A -90.7246323,B 89.1985931,C -90.1231461,S 2,T 2,E1 0.0,E2 0.0,E3 0.0,E4 0.0,E5 0.0,E6 0.0}
DECL LDAT LCPDAT27={VEL 2.00000,ACC 100.000,APO_DIST 500.000,APO_FAC 50.0000,AXIS_VEL 100.000,AXIS_ACC 100.000,ORI_TYP #VAR,CIRC_TYP #BASE,JERK_FAC 50.0000,GEAR_JERK 100.000,EXAX_IGN 0}
DECL E6POS XP33={X 473.022705,Y -91.3580322,Z 290.383667,A -90.7246246,B 89.1985931,C -90.1231308,S 2,T 2,E1 0.0,E2 0.0,E3 0.0,E4 0.0,E5 0.0,E6 0.0}
DECL LDAT LCPDAT28={VEL 2.00000,ACC 100.000,APO_DIST 500.000,APO_FAC 50.0000,AXIS_VEL 100.000,AXIS_ACC 100.000,ORI_TYP #VAR,CIRC_TYP #BASE,JERK_FAC 50.0000,GEAR_JERK 100.000,EXAX_IGN 0}
DECL E6POS XP34={X 473.022705,Y -91.3580322,Z 356.791260,A -90.7246170,B 89.1985931,C -90.1231308,S 2,T 2,E1 0.0,E2 0.0,E3 0.0,E4 0.0,E5 0.0,E6 0.0}
DECL FDAT FP34={TOOL_NO 1,BASE_NO 0,IPO_FRAME #BASE,POINT2[] " "}
DECL LDAT LCPDAT29={VEL 2.00000,ACC 100.000,APO_DIST 500.000,APO_FAC 50.0000,AXIS_VEL 100.000,AXIS_ACC 100.000,ORI_TYP #VAR,CIRC_TYP #BASE,JERK_FAC 50.0000,GEAR_JERK 100.000,EXAX_IGN 0}
ENDDAT
